FUNCTION_BLOCK FB_Blinklicht
VAR_INPUT
	bStartStop	: BOOL;
	tPeriode	: TIME := T#1.5S;
END_VAR
VAR_OUTPUT
	bBlink	:BOOL;
END_VAR
VAR
	fbTon	:Ton;
	fbRtrig	:R_Trig;
	bEinAus	:BOOL;
END_VAR

fbRtrig(CLK:= bStartStop , Q=> );

IF fbRtrig.Q THEN
	bEinAus := NOT bEinAus;
END_IF

//fbTon.IN := bBlink AND NOT fbTon.Q;
//fbTon.PT := T#1S;

fbTon(IN:=bEinAus AND NOT fbTon.Q , PT:=T#1.5S , Q=> , ET=> );


IF fbTon.ET <= fbTon.PT/2 THEN 
	bBlink := FALSE;
ELSIF fbTon.ET > fbTon.PT/2 THEN
	bBlink := TRUE;
END_IF

END_FUNCTION_BLOCK

(* stored: Version 1.1.0.1, ProductVersion 3.1.4024.15
   POU FB_Blinklicht: Id {cf1c7dd2-ae45-498b-93c3-ad3d5f6177a0}, SpecialFunc None *)
